(* CoDeSys 2.3 export: MODULEADDR.EXP *)

(* Data type *)
TYPE ModuleAddr :
(
    A2 := 22,
    A3 := 33,
    A4 := 44,
    A5 := 55,
    A6 := 66,
    A7 := 77
);
END_TYPE
